Staubli VAL3: atan2.pgx

public program atan2(num x_nY, num x_nX, num& x_nResult)
begin
  if x_nX > 0
      x_nResult = atan(x_nY / x_nX)
  elseIf (x_nX < 0) and (x_nY >= 0)
      x_nResult = atan(x_nY / x_nX) + 180.0
  elseIf (x_nX < 0) and (x_nY < 0)
      x_nResult = atan(x_nY / x_nX) - 180.0
  elseIf (x_nX==0) and (x_nY > 0)
      x_nResult = 90.0
  elseIf (x_nX==0) and (x_nY < 0)
      x_nResult = -90.0
  elseIf (x_nX==0) and (x_nY==0)
      x_nResult = 0
  endIf
end
